// TwinCAT 3 PLC project Untitled1
// ProgramVersion: 3.1.4020.1
// libraries:
//   Tc2_EtherCAT, * (Beckhoff Automation GmbH)
//   Tc2_MC2, * (Beckhoff Automation GmbH)
//   Tc2_NCI, * (Beckhoff Automation GmbH)
//   Tc2_Standard, * (Beckhoff Automation GmbH)
//   Tc2_System, * (Beckhoff Automation GmbH)
//   Tc3_Module, * (Beckhoff Automation GmbH)
// project tree:
//   DUTs/ ST_DOX_Control.TcDUT, ST_DOX_STATUS.TcDUT, ST_FastMFunc.TcDUT, ST_MTO_Input.TcDUT, ST_MTO_Outputs.TcDUT, ST_NciChannelFromPlc.TcDUT, ST_NciChannelToPlc.TcDUT
//   / PlcTask.TcTTO
//   POUs/FB_Initialize Axes/ FB_Initialize.TcPOU, ST_Intern_Initialize.TcDUT, ST_PAIn_Initialize.TcDUT, ST_Status_Initialize.TcDUT, ST_Config_Initialize.TcDUT
//   POUs/FB_Valve/ FB_Valve.TcPOU, ST_Config_Valve.TcDUT, ST_PAIn_Valve.TcDUT, ST_PAOut_Valve.TcDUT
//   POUs/FB_Interpreter/ FB_Interpreter.TcPOU, ST_Config_Interpreter.TcDUT, ST_Intern_Interpreter.TcDUT, ST_PAIn_Interpreter.TcDUT, ST_PAOut_Interpreter.TcDUT, ST_Status_Interpreter.TcDUT
//   POUs/POU_Main/ MAIN.TcPOU, ST_Config_Main.TcDUT, ST_Intern_Main.TcDUT, ST_PAIn_Main.TcDUT, ST_PAOut_Main.TcDUT, ST_Status_Main.TcDUT
//   POUs/POU_Drops/ POU_Drops.TcPOU, ST_Config_Drops.TcDUT, ST_PAIn_Drops.TcDUT, ST_PAOut_Drops.TcDUT
// real-time tasks:
//   TASK PlcTask: cycle T#10ms, priority 20, ADS port 350
// motion (NC):
//   TASK NC-Task 1 SAF: cycle T#2ms, priority 4, ADS port 501
//   TASK NC-Task 1 SVB: cycle T#10ms, priority 8, ADS port 511
//   AXIS Axis 1 (id 1)
//     Dynamic: AccelerationMaximum=700, DecelerationMaximum=700, Acceleration=632.077, Deceleration=632.077, Jerk=142686, DelayTime=0.008, OverrideType=4
//     Velo: RefSync=5, SlowManual=25, FastManual=50, Fast=50, Maximum=280
//     PositionAreaControl: Enable=false, RefSearch=false
//     TargetPosControl: Enable=false
//     OtherSettings: AllowMotionCmdToSlave=true
//     encoder EncType=4
//       EncPara: ScaleFactorNumerator=0.002334, MaxCount=#x0000ffff
//         ActPosCorrection: Time=0.02
//         Inc: RefSearchInverse=true, RefSyncInverse=false, RefMode=1, RefSoftSyncMask=#x0000ffff
//     drive DrvType=24
//       Analog: VeloReferenz=300
//       TimeComp: TaskDelayCycles=1
//     controller CtrType=2
//       CtrPara: PriorControlFactor=1
//         PosDiffControl: Enable=false
//         PID: PosKp=100, PosExtKp=100, DeadBandPosition=0.01
//         Observer: BandWidth=20
//   AXIS Axis 2 (id 2)
//     Dynamic: AccelerationMaximum=700, DecelerationMaximum=700, Acceleration=632.077, Deceleration=632.077, Jerk=142686, DelayTime=0.008, OverrideType=4
//     Velo: RefSync=5, SlowManual=25, FastManual=50, Fast=50, Maximum=280
//     PositionAreaControl: Enable=false, RefSearch=false
//     TargetPosControl: Enable=false
//     OtherSettings: AllowMotionCmdToSlave=true
//     encoder EncType=4
//       EncPara: ScaleFactorNumerator=0.002334, MaxCount=#x0000ffff
//         ActPosCorrection: Time=0.02
//         Inc: RefSearchInverse=true, RefSyncInverse=false, RefMode=1, RefSoftSyncMask=#x0000ffff
//     drive DrvType=24
//       Analog: VeloReferenz=300
//       TimeComp: TaskDelayCycles=1
//     controller CtrType=2
//       CtrPara: PriorControlFactor=1
//         PosDiffControl: Enable=false
//         PID: PosKp=100, PosExtKp=100, DeadBandPosition=0.01
//         Observer: BandWidth=20
// I/O:
//   DEVICE Device 2 (EtherCAT), AmsNetId 192.168.31.63.3.1
//     Term 1 (EK1101) [EK1101 EtherCAT Coupler (2A E-Bus, ID switch)]
//       Term 2 (EL2008) [EL2008 8Ch. Dig. Output 24V, 0.5A]
//       Term 3 (EL7037) [EL7037 1Ch. Stepper motor output stage (24V, 1.5A)]
//       Term 4 (EL7037) [EL7037 1Ch. Stepper motor output stage (24V, 1.5A)]
//       Term 5 (EL1018) [EL1018 8Ch. Dig. Input 24V, 10µs]
//       Term 6 (EL4004) [EL4004 4Ch. Ana. Output 0-10V, 12bit]
//       Term 7 (EL3064) [EL3064 4Ch. Ana. Input 0-10V]
//       Term 8 (EL3318) [EL3318 8Ch. Ana Input Thermocouple (TC)]
//       Term 9 (EL9576) [EL9576 Brake chopper terminal]
//       Term 10 (EL2212) [EL2212 2Ch. dig. output with overexcitation (24V DC, 2.5A, 10A Peak)]
//       Term 11 (EL9011) [EL9011 End Terminal]
// variable links:
//   NC-Task 1 SAF/Axes/Axis 1 <-> Device 2 (EtherCAT)/Term 1 (EK1101)/Term 3 (EL7037)
//     Drive/Inputs/In/nState1 @bit 3 <-> STM Status/Status/Error
//     Drive/Inputs/In/nState1 @bit 7 <-> STM Status/Status/Motor stall
//     Drive/Inputs/In/nState1 @bit 5 <-> STM Status/Status/Moving negative
//     Drive/Inputs/In/nState1 @bit 4 <-> STM Status/Status/Moving positive
//     Drive/Inputs/In/nState1 @bit 1 <-> STM Status/Status/Ready
//     Drive/Inputs/In/nState1 <-> STM Status/Status/Ready to enable
//     Drive/Inputs/In/nState1 @bit 6 <-> STM Status/Status/Torque reduced
//     Drive/Inputs/In/nState1 @bit 2 <-> STM Status/Status/Warning
//     Drive/Inputs/In/nState2 @bit 3 <-> STM Status/Status/Digital input 1
//     Drive/Inputs/In/nState2 @bit 4 <-> STM Status/Status/Digital input 2
//     Drive/Inputs/In/nState2 @bit 5 <-> STM Status/Status/Sync error
//     Drive/Inputs/In/nState2 @bit 7 <-> STM Status/Status/TxPDO Toggle
//     Drive/Inputs/In/nState4 @bit 1 <-> WcState/InputToggle
//     Drive/Inputs/In/nState4 <-> WcState/WcState
//     Drive/Outputs/Out/nCtrl1 <-> STM Control/Control/Enable
//     Drive/Outputs/Out/nCtrl1 @bit 2 <-> STM Control/Control/Reduce torque
//     Drive/Outputs/Out/nCtrl1 @bit 1 <-> STM Control/Control/Reset
//     Drive/Outputs/Out/nCtrl2 @bit 3 <-> STM Control/Control/Digital output 1
//     Drive/Outputs/Out/nDataOut2[0] <-> STM Velocity/Velocity
//     Enc/Inputs/In/nDataIn1[0] <-> ENC Status compact/Counter value
//     Enc/Inputs/In/nDataIn2[0] <-> ENC Status compact/Latch value
//     Enc/Inputs/In/nState1 @bit 4 <-> ENC Status compact/Status/Counter overflow
//     Enc/Inputs/In/nState1 @bit 3 <-> ENC Status compact/Status/Counter underflow
//     Enc/Inputs/In/nState1 @bit 7 <-> ENC Status compact/Status/Extrapolation stall
//     Enc/Inputs/In/nState1 <-> ENC Status compact/Status/Latch C valid
//     Enc/Inputs/In/nState1 @bit 1 <-> ENC Status compact/Status/Latch extern valid
//     Enc/Inputs/In/nState1 @bit 2 <-> ENC Status compact/Status/Set counter done
//     Enc/Inputs/In/nState2 @bit 4 <-> ENC Status compact/Status/Status of extern latch
//     Enc/Inputs/In/nState2 <-> ENC Status compact/Status/Status of input A
//     Enc/Inputs/In/nState2 @bit 1 <-> ENC Status compact/Status/Status of input B
//     Enc/Inputs/In/nState2 @bit 2 <-> ENC Status compact/Status/Status of input C
//     Enc/Inputs/In/nState2 @bit 5 <-> ENC Status compact/Status/Sync error
//     Enc/Inputs/In/nState2 @bit 7 <-> ENC Status compact/Status/TxPDO Toggle
//     Enc/Inputs/In/nState4 @bit 1 <-> WcState/InputToggle
//     Enc/Inputs/In/nState4 <-> WcState/WcState
//     Enc/Outputs/Out/nCtrl1 <-> ENC Control compact/Control/Enable latch C
//     Enc/Outputs/Out/nCtrl1 @bit 3 <-> ENC Control compact/Control/Enable latch extern on negative edge
//     Enc/Outputs/Out/nCtrl1 @bit 1 <-> ENC Control compact/Control/Enable latch extern on positive edge
//     Enc/Outputs/Out/nCtrl1 @bit 2 <-> ENC Control compact/Control/Set counter
//     Enc/Outputs/Out/nDataOut1[0] <-> ENC Control compact/Set counter value
//   NC-Task 1 SAF/Axes/Axis 2 <-> Device 2 (EtherCAT)/Term 1 (EK1101)/Term 4 (EL7037)
//     Drive/Inputs/In/nState1 @bit 3 <-> STM Status/Status/Error
//     Drive/Inputs/In/nState1 @bit 7 <-> STM Status/Status/Motor stall
//     Drive/Inputs/In/nState1 @bit 5 <-> STM Status/Status/Moving negative
//     Drive/Inputs/In/nState1 @bit 4 <-> STM Status/Status/Moving positive
//     Drive/Inputs/In/nState1 @bit 1 <-> STM Status/Status/Ready
//     Drive/Inputs/In/nState1 <-> STM Status/Status/Ready to enable
//     Drive/Inputs/In/nState1 @bit 6 <-> STM Status/Status/Torque reduced
//     Drive/Inputs/In/nState1 @bit 2 <-> STM Status/Status/Warning
//     Drive/Inputs/In/nState2 @bit 3 <-> STM Status/Status/Digital input 1
//     Drive/Inputs/In/nState2 @bit 4 <-> STM Status/Status/Digital input 2
//     Drive/Inputs/In/nState2 @bit 5 <-> STM Status/Status/Sync error
//     Drive/Inputs/In/nState2 @bit 7 <-> STM Status/Status/TxPDO Toggle
//     Drive/Inputs/In/nState4 @bit 1 <-> WcState/InputToggle
//     Drive/Inputs/In/nState4 <-> WcState/WcState
//     Drive/Outputs/Out/nCtrl1 <-> STM Control/Control/Enable
//     Drive/Outputs/Out/nCtrl1 @bit 2 <-> STM Control/Control/Reduce torque
//     Drive/Outputs/Out/nCtrl1 @bit 1 <-> STM Control/Control/Reset
//     Drive/Outputs/Out/nCtrl2 @bit 3 <-> STM Control/Control/Digital output 1
//     Drive/Outputs/Out/nDataOut2[0] <-> STM Velocity/Velocity
//     Enc/Inputs/In/nDataIn1[0] <-> ENC Status compact/Counter value
//     Enc/Inputs/In/nDataIn2[0] <-> ENC Status compact/Latch value
//     Enc/Inputs/In/nState1 @bit 4 <-> ENC Status compact/Status/Counter overflow
//     Enc/Inputs/In/nState1 @bit 3 <-> ENC Status compact/Status/Counter underflow
//     Enc/Inputs/In/nState1 @bit 7 <-> ENC Status compact/Status/Extrapolation stall
//     Enc/Inputs/In/nState1 <-> ENC Status compact/Status/Latch C valid
//     Enc/Inputs/In/nState1 @bit 1 <-> ENC Status compact/Status/Latch extern valid
//     Enc/Inputs/In/nState1 @bit 2 <-> ENC Status compact/Status/Set counter done
//     Enc/Inputs/In/nState2 @bit 4 <-> ENC Status compact/Status/Status of extern latch
//     Enc/Inputs/In/nState2 <-> ENC Status compact/Status/Status of input A
//     Enc/Inputs/In/nState2 @bit 1 <-> ENC Status compact/Status/Status of input B
//     Enc/Inputs/In/nState2 @bit 2 <-> ENC Status compact/Status/Status of input C
//     Enc/Inputs/In/nState2 @bit 5 <-> ENC Status compact/Status/Sync error
//     Enc/Inputs/In/nState2 @bit 7 <-> ENC Status compact/Status/TxPDO Toggle
//     Enc/Inputs/In/nState4 @bit 1 <-> WcState/InputToggle
//     Enc/Inputs/In/nState4 <-> WcState/WcState
//     Enc/Outputs/Out/nCtrl1 <-> ENC Control compact/Control/Enable latch C
//     Enc/Outputs/Out/nCtrl1 @bit 3 <-> ENC Control compact/Control/Enable latch extern on negative edge
//     Enc/Outputs/Out/nCtrl1 @bit 1 <-> ENC Control compact/Control/Enable latch extern on positive edge
//     Enc/Outputs/Out/nCtrl1 @bit 2 <-> ENC Control compact/Control/Set counter
//     Enc/Outputs/Out/nDataOut1[0] <-> ENC Control compact/Set counter value
//   Untitled1/Untitled1 Instance <-> Device 2 (EtherCAT)/Term 1 (EK1101)/Term 10 (EL2212)
//     PlcTask Inputs/MAIN.stPAIn/stPAInDrops/stValve/stDOXStatus1/bError <-> DOX Status (MTO) Channel 1/Status/Error
//     PlcTask Inputs/MAIN.stPAIn/stPAInDrops/stValve/stDOXStatus1/bPWMActive <-> DOX Status (MTO) Channel 1/Status/PWM active
//     PlcTask Inputs/MAIN.stPAIn/stPAInDrops/stValve/stDOXStatus1/bReadyToActivate <-> DOX Status (MTO) Channel 1/Status/Ready to activate
//     PlcTask Inputs/MAIN.stPAIn/stPAInDrops/stValve/stDOXStatus1/bTxPDO <-> DOX Status (MTO) Channel 1/Status/TxPDO Toggle
//     PlcTask Inputs/MAIN.stPAIn/stPAInDrops/stValve/stDOXStatus1/bWarning <-> DOX Status (MTO) Channel 1/Status/Warning
//     PlcTask Inputs/MAIN.stPAIn/stPAInDrops/stValve/stMTOInputs1/b2InputCycleCounter <-> MTO Inputs Channel 1/Status/Input cycle counter
//     PlcTask Inputs/MAIN.stPAIn/stPAInDrops/stValve/stMTOInputs1/bOutputBufferOverflow <-> MTO Inputs Channel 1/Status/Output buffer overflow
//     PlcTask Inputs/MAIN.stPAIn/stPAInDrops/stValve/stMTOInputs1/bOutputShortCircuit <-> MTO Inputs Channel 1/Status/Output short circuit
//     PlcTask Inputs/MAIN.stPAIn/stPAInDrops/stValve/stMTOInputs1/bOutputState <-> MTO Inputs Channel 1/Status/Output state
//     PlcTask Inputs/MAIN.stPAIn/stPAInDrops/stValve/stMTOInputs1/bWarning <-> MTO Inputs Channel 1/Status/Warning
//     PlcTask Inputs/MAIN.stPAIn/stPAInDrops/stValve/stMTOInputs1/iEventsInOutput <-> MTO Inputs Channel 1/Status/Events in output buffer
//     PlcTask Inputs/MAIN.stPAIn/stPAInDrops/stValve/stMTOInputs1/iOutputOrderFeedback <-> MTO Inputs Channel 1/Status/Output order feedback
//     PlcTask Outputs/MAIN.stPAOut/stPAOutDrops/stValve/stDoxControl1/bPWM <-> DOX Control (MTO) Channel 1/Control/PWM
//     PlcTask Outputs/MAIN.stPAOut/stPAOutDrops/stValve/stDoxControl1/bReset <-> DOX Control (MTO) Channel 1/Control/Reset
//     PlcTask Outputs/MAIN.stPAOut/stPAOutDrops/stValve/stMTOOutputs1/bBufferReset <-> MTO Outputs 2x Channel 1/Ctrl/Output buffer reset
//     PlcTask Outputs/MAIN.stPAOut/stPAOutDrops/stValve/stMTOOutputs1/bEnableManualOp <-> MTO Outputs 2x Channel 1/Ctrl/Enable manual operation
//     PlcTask Outputs/MAIN.stPAOut/stPAOutDrops/stValve/stMTOOutputs1/bForceOrder <-> MTO Outputs 2x Channel 1/Ctrl/Force order
//     PlcTask Outputs/MAIN.stPAOut/stPAOutDrops/stValve/stMTOOutputs1/bManualOutputState <-> MTO Outputs 2x Channel 1/Ctrl/Manual output state
//     PlcTask Outputs/MAIN.stPAOut/stPAOutDrops/stValve/stMTOOutputs1/bOutputEventState1 <-> MTO Outputs 2x Channel 1/Outputs/Output event state 1
//     PlcTask Outputs/MAIN.stPAOut/stPAOutDrops/stValve/stMTOOutputs1/bOutputEventState2 <-> MTO Outputs 2x Channel 1/Outputs/Output event state 2
//     PlcTask Outputs/MAIN.stPAOut/stPAOutDrops/stValve/stMTOOutputs1/iNoOfOutputEvents <-> MTO Outputs 2x Channel 1/Ctrl/No of output events
//     PlcTask Outputs/MAIN.stPAOut/stPAOutDrops/stValve/stMTOOutputs1/iOutputOrderCount <-> MTO Outputs 2x Channel 1/Ctrl/Output order counter
//     PlcTask Outputs/MAIN.stPAOut/stPAOutDrops/stValve/stMTOOutputs1/tOutputEventTime1 <-> MTO Outputs 2x Channel 1/Output event time 1
//     PlcTask Outputs/MAIN.stPAOut/stPAOutDrops/stValve/stMTOOutputs1/tOutputEventTime2 <-> MTO Outputs 2x Channel 1/Output event time 2
//   Untitled1/Untitled1 Instance <-> Device 2 (EtherCAT)/Term 1 (EK1101)/Term 3 (EL7037)
//     PlcTask Inputs/MAIN.stPAIn/stInit/bXCam <-> STM Status/Status/Digital input 1
//   Untitled1/Untitled1 Instance <-> Device 2 (EtherCAT)/Term 1 (EK1101)/Term 4 (EL7037)
//     PlcTask Inputs/MAIN.stPAIn/stInit/bYCam <-> STM Status/Status/Digital input 1
//   Untitled1/Untitled1 Instance <-> NC-Task 1 SAF/Axes/Axis 1
//     PlcTask Inputs/MAIN.fbInitialize.XAxis.NcToPlc <-> Outputs/ToPlc
//     PlcTask Outputs/MAIN.fbInitialize.XAxis.PlcToNc <-> Inputs/FromPlc
//   Untitled1/Untitled1 Instance <-> NC-Task 1 SAF/Axes/Axis 2
//     PlcTask Inputs/MAIN.fbInitialize.YAxis.NcToPlc <-> Outputs/ToPlc
//     PlcTask Outputs/MAIN.fbInitialize.YAxis.PlcToNc <-> Inputs/FromPlc
//   Untitled1/Untitled1 Instance <-> NC-Task 1 SAF/Channel 2
//     PlcTask Inputs/MAIN.stPAIn/stInterp/in_stItpToPlc <-> Outputs/ToPlc
//     PlcTask Inputs/MAIN.stPAIn/stMBits <-> Outputs/ToPlc/FastMFuncMask[1]
//     PlcTask Outputs/MAIN.stPAOut/stInterp/out_stPlcToItp <-> Inputs/FromPlc

CONFIGURATION Untitled1
    RESOURCE PLC ON TwinCAT3
        TASK PlcTask(INTERVAL := T#10ms, PRIORITY := 20);
        PROGRAM MAIN WITH PlcTask : MAIN;
    END_RESOURCE
END_CONFIGURATION

// ---- DUTs/ST_DOX_Control.TcDUT
TYPE ST_DOX_Control :
STRUCT
	bBit0    :				BIT;	//71.0
	bBit1    :				BIT;
	bBit2    :				BIT;
	bPWM  :					BIT:=1;	//71.3
	bBit4  :				BIT;
	bBit5  :				BIT;
	bBit6  :				BIT;
	bReset  :				BIT;	//71.7
	BByte8   :				BYTE;
	
END_STRUCT
END_TYPE

// ---- DUTs/ST_DOX_STATUS.TcDUT
TYPE ST_DOX_STATUS :
STRUCT
	bReadyToActivate:	BIT;
	bPWMActive:			BIT;
	bWarning:			BIT;
	bError:				BIT;
	bTxPDO:				BIT;
END_STRUCT
END_TYPE

// ---- DUTs/ST_FastMFunc.TcDUT
TYPE ST_FastMFunc :
STRUCT
	bMbit0:			BIT;
	bMBit1:			BIT;
	bMBit2:			BIT;
	bMBit3:			BIT;
	bMBit4:			BIT;
	bMBit5:			BIT;
	bMBit6:			BIT;
	bMBit7:			BIT;
	bMBit8:			BIT;
	bMBit9:			BIT;
	bMBit10:		BIT;
	bMBit11:		BIT;
	bMBit12:		BIT;
	bMBit13:		BIT;
	bMBit14:		BIT;
	bMBit15:		BIT;
	bMBit16:		BIT;
	bMBit17:		BIT;
	bMBit18:		BIT;
	bMBit19:		BIT;
	bMBit20:		BIT;
	bMBit21:		BIT;
	bMBit22:		BIT;
	bMBit23:		BIT;
	bMBit24:		BIT;
	bMBit25:		BIT;
	bMBit26:		BIT;
	bMBit27:		BIT;
	bMBit28:		BIT;
	bMBit29:		BIT;
	bMBit30:		BIT;
	bMBit31:		BIT;	
END_STRUCT
END_TYPE

// ---- DUTs/ST_MTO_Input.TcDUT
TYPE ST_MTO_Input :
STRUCT
	bOutputShortCircuit:			BOOL;
	bOutputBufferOverflow:			BOOL;
	bOutputState:					BOOL;
	bWarning:						BOOL;
	b2InputCycleCounter:			BOOL;
	iOutputOrderFeedback:			USINT;
	iEventsInOutput:				USINT;
END_STRUCT
END_TYPE

// ---- DUTs/ST_MTO_Outputs.TcDUT
TYPE ST_MTO_Outputs :
STRUCT
	
	bBufferReset    :				BIT;	//73.0
	bManualOutputState    :			BIT;
	bForceOrder    :				BIT:=1;
	bEnableManualOp  :				BIT;	//73.3
	bBit4  :						BIT;
	bBit5  :						BIT;
	bBit6  :						BIT;
	bBit7  :						BIT;
	iOutputOrderCount  :			USINT;	//74.0
	iNoOfOutputEvents  :			USINT;	//75.0
	Bbyte24:						BYTE;
	bOutputEventState1	:			BIT;
	bOutputEventState2	:			BIT;
	tOutputEventTime1:				UDINT;
	tOutputEventTime2:				UDINT;
END_STRUCT
END_TYPE

// ---- DUTs/ST_NciChannelFromPlc.TcDUT
TYPE ST_NciChannelFromPlc :
STRUCT
    nSkipLine        : WORD; (* Mask to skip lines *)
    nItpMode         : WORD;
    nMFuncGranted    : WORD; (* granted signal of the M-function *)
    nReserved1       : ARRAY[7..8] OF BYTE;
    nChaAxesOvr      : DWORD; (* Channel override in percent * 100 *)
    nChaSpindleOvr   : DWORD;
    nReserved2       : ARRAY[17..128] OF BYTE;
END_STRUCT
END_TYPE

// ---- DUTs/ST_NciChannelToPlc.TcDUT
TYPE ST_NciChannelToPlc :
STRUCT
	
    nJobNo         : DWORD;
    nFastMFuncMask : ARRAY[1..5] OF DWORD; (* Mask to evaluate fast M-functions *)
    nHskMFuncNo    : WORD; (* evaluate M-function with handshake *)
    nHskMFuncReq   : WORD;
    nHFuncValue    : DINT;
    nSpindleRpm    : WORD;
    nTool          : WORD;
    nReserved1     : ARRAY[37..132] OF BYTE;
    nLoadedProg    : DWORD; (* loaded program number if exist *)
    nItpMode       : WORD; (* Interpreter mode *)
    nItpState      : WORD; (* Interpreter status *)
    nItpErrCode    : UDINT; (* Interpreter-Channel Error Code Changed from *WORD*)
    nReserved2     : ARRAY[143..150] OF BYTE;
	
END_STRUCT
END_TYPE

// ---- POUs/FB_Initialize Axes/ST_Intern_Initialize.TcDUT
TYPE ST_Intern_Initialize :
STRUCT
		tnReady		:TON;
		
END_STRUCT
END_TYPE

// ---- POUs/FB_Initialize Axes/ST_PAIn_Initialize.TcDUT
TYPE ST_PAIn_Initialize :
STRUCT
	
(*Homing Notches*)	
	bXCam	:BOOL;  	
	bYCam	:BOOL;
	
END_STRUCT
END_TYPE

// ---- POUs/FB_Initialize Axes/ST_Status_Initialize.TcDUT
TYPE ST_Status_Initialize :
STRUCT
	bFini	:BOOL;
	bBus	:BOOL;
	bErr	:BOOL;
	nErr	:UDINT;
	iItpState:	UDINT;
	iState: INT;
END_STRUCT
END_TYPE

// ---- POUs/FB_Initialize Axes/ST_Config_Initialize.TcDUT
TYPE ST_Config_Initialize :
STRUCT
	nXA					:UDINT:=1;
	nYA					:UDINT:=2;
	nZA					:UDINT:=0;
	nGroup				:UDINT:=3;
	tTimeO				:TIME:=T#5S;
	g_strProgram		:STRING := 'C:\Users\Furkan\Desktop\FirstNciSample\TestIt.nc';
	bExe				:BOOL:=TRUE;
	bSta				:BOOL:=TRUE;
	bSto				:BOOL:=FALSE;
	
END_STRUCT
END_TYPE

// ---- POUs/FB_Valve/ST_Config_Valve.TcDUT
TYPE ST_Config_Valve:
STRUCT
END_STRUCT
END_TYPE

// ---- POUs/FB_Valve/ST_PAIn_Valve.TcDUT
TYPE ST_PAIn_Valve :
STRUCT
	stDOXStatus1: ST_DOX_STATUS;
	
	stMTOInputs1: ST_MTO_Input;
	
	
	

END_STRUCT
END_TYPE

// ---- POUs/FB_Valve/ST_PAOut_Valve.TcDUT
TYPE ST_PAOut_Valve :
STRUCT
	stMTOOutputs1:			ST_MTO_Outputs;
	stDoxControl1:			ST_DOX_Control;
	
	
	
END_STRUCT
END_TYPE

// ---- POUs/FB_Interpreter/ST_Config_Interpreter.TcDUT
TYPE ST_Config_Interpreter :
STRUCT
	bInit				:BOOL;
	nXA					:UDINT:=1;
	nYA					:UDINT:=2;
	nZA					:UDINT:=0;
	nGroup				:UDINT:=3;
	tTimeO				:TIME:=T#5S;
	g_strProgram		:STRING := 'D:\Semester\NC.nc';
	bExe				:BOOL:=TRUE;
	bSta				:BOOL:=TRUE;
	bSto				:BOOL:=FALSE;
	
END_STRUCT
END_TYPE

// ---- POUs/FB_Interpreter/ST_Intern_Interpreter.TcDUT
TYPE ST_Intern_Interpreter :
STRUCT
	
		
END_STRUCT
END_TYPE

// ---- POUs/FB_Interpreter/ST_PAIn_Interpreter.TcDUT
TYPE ST_PAIn_Interpreter :
STRUCT

		in_stItpToPlc			:NCTOPLC_NCICHANNEL_REF;
	
END_STRUCT
END_TYPE

// ---- POUs/FB_Interpreter/ST_PAOut_Interpreter.TcDUT
TYPE ST_PAOut_Interpreter :
STRUCT
	
	
	out_stPlcToItp			:PLCTONC_NCICHANNEL_REF;	
END_STRUCT
END_TYPE

// ---- POUs/FB_Interpreter/ST_Status_Interpreter.TcDUT
TYPE ST_Status_Interpreter :
STRUCT
	bFini	:BOOL;
	bBus	:BOOL;
	bErr	:BOOL;
	nErr	:UDINT;
	iItpState:	UDINT;
	iState: INT;
END_STRUCT
END_TYPE

// ---- POUs/POU_Main/ST_Config_Main.TcDUT
TYPE ST_Config_Main :
STRUCT
	
	stInterp			:ST_Config_Interpreter;
	stInit				:ST_Config_Initialize;
END_STRUCT
END_TYPE

// ---- POUs/POU_Main/ST_Intern_Main.TcDUT
TYPE ST_Intern_Main :
STRUCT
	count: INT;
	
END_STRUCT
END_TYPE

// ---- POUs/POU_Main/ST_PAIn_Main.TcDUT
TYPE ST_PAIn_Main :
STRUCT
	(* stNcToPlc	:ST_NciChannelToPlc;  
	stNciIn		:ST_NCInterpreter_PAIn;*)

	stInit			:ST_PAIn_Initialize;
	stInterp		:ST_PAIn_Interpreter;
	stMBits			:ST_FastMFunc;
	stPAInDrops		:ST_PAIn_Drops;
	

END_STRUCT
END_TYPE

// ---- POUs/POU_Main/ST_PAOut_Main.TcDUT
TYPE ST_PAOut_Main :
STRUCT
	
	stInterp					:ST_PAOut_Interpreter;
	stPAOutDrops				:ST_PAOut_Drops;
END_STRUCT
END_TYPE

// ---- POUs/POU_Main/ST_Status_Main.TcDUT
TYPE ST_Status_Main :
STRUCT
	stInterp				:ST_Status_Interpreter;
	stInit					:ST_Status_Initialize;
END_STRUCT
END_TYPE

// ---- POUs/POU_Drops/ST_Config_Drops.TcDUT
TYPE ST_Config_Drops :
STRUCT
	stValve: ST_Config_Valve;
	
END_STRUCT
END_TYPE

// ---- POUs/POU_Drops/ST_PAIn_Drops.TcDUT
TYPE ST_PAIn_Drops :
STRUCT
	stValve 			:ST_PAIn_Valve;
	
END_STRUCT
END_TYPE

// ---- POUs/POU_Drops/ST_PAOut_Drops.TcDUT
TYPE ST_PAOut_Drops :
STRUCT
	stValve: ST_PAOut_Valve;
	
END_STRUCT
END_TYPE

// ---- POUs/POU_Main/MAIN.TcPOU
PROGRAM MAIN

VAR
	stIntern			:ST_Intern_Main;
	fbInitialize		:FB_Initialize;
	fbInterpreter		:FB_Interpreter;
	stStatus			:ST_Status_Main;
	iState				:INT;
END_VAR

VAR_INPUT
	stConfig			:ST_Config_Main;
	stPAIn	AT%I*		:ST_PAIn_Main;
	
END_VAR

VAR_OUTPUT
	stPAOut	AT%Q*		:ST_PAOut_Main;
	
END_VAR

fbInitialize(stPAIn:=stPAIn.stInit,
			stConfig:=stConfig.stInit,
			stStatus=>stStatus.stInit	);


fbInterpreter(stConfig:=stConfig.stInterp,
				stPAOut=>stPAOut.stInterp,
				stStatus=>stStatus.stInterp);

fbInterpreter.stPAIn.in_stItpToPlc:=stPAIn.stInterp.in_stItpToPlc;	


CASE iState OF
	
		00: fbInitialize.bExec:=TRUE;
	
		IF NOT fbInitialize.bBus THEN
			IF fbInitialize.bFini THEN 
				iState:=10;
			END_IF
		END_IF
		
		10: fbInterpreter.bExec:=TRUE;
	
		IF NOT fbInterpreter.bBus THEN
			IF fbInterpreter.bFini THEN 
				iState:=20;
			END_IF
		END_IF
		
	
END_CASE

END_PROGRAM

// ---- POUs/FB_Initialize Axes/FB_Initialize.TcPOU
FUNCTION_BLOCK FB_Initialize
VAR_INPUT
	stPAIn	 				:ST_PAIn_Initialize;
	stConfig				:ST_Config_Initialize;
	bExec				:BOOL;
END_VAR
	
VAR_OUTPUT
	bFini	:BOOL;
	bBus	:BOOL;
	bErr	:BOOL;

	stStatus				:ST_Status_Initialize;
END_VAR

VAR
	stIntern				:ST_Intern_Initialize;
	(*Axis References*)
	XAxis					:AXIS_REF;
	YAxis					:AXIS_REF;
	(*Motion Control Definitions*)
	fbPower_X				:MC_Power;
	fbPower_Y				:MC_Power;
	fbHome_X				:MC_Home;
	fbHome_Y				:MC_Home;
	fbBuildGrp				:CfgBuildExt3DGroup;
END_VAR


XAxis.ReadStatus();
YAxis.ReadStatus();
fbPower_X(Axis:=XAxis);
fbPower_Y(Axis:=YAxis);	
fbHome_X(Axis:=XAxis);
fbHome_Y(Axis:=YAxis);	

CASE stStatus.iState OF 

	00:	IF bExec THEN
			bBus:=TRUE;
 			stStatus.iState:=05;
		END_IF
		

05:
(*Enable X-Axis*)
		fbPower_X.Enable			:=TRUE;
		fbPower_X.Enable_Positive	:=TRUE;
		fbPower_X.Enable_Negative	:=TRUE;
		
(*Enable Y-Axis*)

		fbPower_Y.Enable			:=TRUE;
		fbPower_Y.Enable_Positive	:=TRUE;
		fbPower_Y.Enable_Negative	:=TRUE;
		
	stIntern.tnReady(IN:=fbPower_X.Status AND fbPower_Y.Status,PT:=T#100MS);
			
		IF stIntern.tnReady.Q THEN
			stStatus.iState:=10;
		END_IF
10:	(*Home X-Axis*)
		fbHome_X.HomingMode			:=MC_DefaultHoming;
		fbHome_X.bCalibrationCam	:=stPAIn.bXCam;
		fbHome_X.Execute			:= stConfig.bExe;
		fbHome_X.Position			:= 0;
	(*Home Y-Axis*)
		fbHome_Y.HomingMode			:=MC_DefaultHoming;
		fbHome_Y.bCalibrationCam	:=stPAIn.bYCam;
		fbHome_Y.Execute			:= stConfig.bExe;
		fbHome_Y.Position			:= 0;
		
		IF NOT fbHome_X.Error AND NOT fbHome_Y.Error AND fbHome_X.Done AND fbHome_Y.Done THEN
			stStatus.iState:=20;
		END_IF
		
20:	(* Build group for interpolation*)
		fbBuildGrp	(
		bExecute	:= TRUE ,
		nGroupId	:= stConfig.nGroup,
		nXAxisId	:= stConfig.nXA,
		nYAxisId	:= stConfig.nYA,
		nZAxisId	:= stConfig.nZA,
		nQ1AxisId	:= 0,
		nQ2AxisId	:= 0,
		nQ3AxisId	:= 0,
		nQ4AxisId	:= 0,
		nQ5AxisId	:= 0,
		tTimeOut	:= T#200MS,
		bErr		=>stStatus.bErr,
		bBusy		=>stStatus.bBus,
		nErrId		=>stStatus.nErr);	
				
	stIntern.tnReady(IN:=TRUE AND NOT stStatus.bErr ,PT:=T#2S);
	IF stIntern.tnReady.Q THEN
		bFini:=TRUE;
		bBus:=FALSE;
		stStatus.iState:=30;
	END_IF		

END_CASE

END_FUNCTION_BLOCK

// ---- POUs/FB_Interpreter/FB_Interpreter.TcPOU
FUNCTION_BLOCK FB_Interpreter
VAR
	fbLoadProg				:ItpLoadProgEx;
	fbStart					:ItpStartStopEx;
END_VAR
VAR_INPUT
	bExec					:BOOL;
	stPAIn					:ST_PAIn_Interpreter;
	stConfig				:ST_Config_Interpreter;
END_VAR
VAR_OUTPUT
	bFini	:BOOL;
	bBus	:BOOL;
	bErr	:BOOL;

	stPAOut					:ST_PAOut_Interpreter;
	stStatus				:ST_Status_Interpreter;
END_VAR

CASE stStatus.iState OF
		

	00: IF 	bExec THEN
			bBus:=TRUE;
			stStatus.iState:=05;
		END_IF


	05:
		fbLoadProg(
		bExecute	:= TRUE,
		sPrg		:= stConfig.g_strProgram,
		nLength		:= LEN(stConfig.g_strProgram),
		tTimeOut	:= T#200MS,
		sNciToPlc	:= MAIN.stPAIn.stInterp.in_stItpToPlc);
		
	stStatus.iItpState		:=	ItpGetStateInterpreter(stPAIn.in_stItpToPlc );
	
	IF stStatus.iItpState = NCI_INTERPRETER_READY THEN
		(* load part program succeeded *)
		stStatus.iState	:= 10;
	ELSIF stStatus.iItpState = NCI_INTERPRETER_ABORTED THEN
		(* load program failed - probably there is a load time error, e.g. syntax error *)
		(* add error handling here *)
		stStatus.bErr		:= TRUE;
		stStatus.nErr	:= 4711;	(* substitute with own error code *)
		stStatus.iState	:= 200;
	END_IF
	
	10: ItpSetOverridePercent( fOverridePercent:=100, sPlcToNci:=stPAOut.out_stPlcToItp );
	
		fbStart(
				bStart		:= stConfig.bSta,
				bStop		:= stConfig.bSto,
				tTimeOut	:= T#200MS,
				sNciToPlc	:=Main.stPAIn.stInterp.in_stItpToPlc
				);

	IF NOT fbStart.bBusy THEN
		fbStart( bStart:=FALSE, sNciToPlc:=stPAIn.in_stItpToPlc );
		IF NOT fbStart.bErr THEN
			stStatus.iState	:= 20;
		ELSE
			(* an error occured *)
			stStatus.bErr		:= TRUE;
			stStatus.nErr	:= fbStart.nErrId;
			stStatus.iState	:= 200;
		END_IF
	END_IF
		
	20:	stStatus.iItpState	:=	ItpGetStateInterpreter(  sNciToPlc:=MAIN.stPAIn.stInterp.in_stItpToPlc );
	IF stStatus.iItpState <> NCI_INTERPRETER_READY THEN
		bFini:=TRUE;
		bBus:=FALSE;
		stStatus.iState	:= 40;
	END_IF
				
END_CASE

END_FUNCTION_BLOCK

// ---- POUs/FB_Valve/FB_Valve.TcPOU
FUNCTION_BLOCK FB_Valve
VAR_INPUT
	
	stConfig:	ST_Config_Valve;
	stPAIn	:	ST_PAIn_Valve;
	
	iPeriod: 	UDINT:= 40000000;
	tPeriod: 	TIME;
	iDuration: 	UDINT:= 9000000;
	bActivate: 	BOOL:=TRUE;
	
END_VAR
VAR_OUTPUT
	stPAOut	:	ST_PAOut_Valve;
END_VAR
	
VAR
	iEvent1: 		UDINT;
	iEvent2:		UDINT;	
	nNoOfOutputEvents: INT;
	nOutputOrderCnt: USINT;
	
	tnHalt: 			TON;
 	iCurrentTime:  	ULINT;
 	iCurrentTime32:  	UDINT;
	
	nScheduleNo: INT;
	iState:			UINT:=0;
	iLastTime: UDINT;
END_VAR

	iCurrentTime := F_GetCurDcTaskTime64();
	iCurrentTime32:=ULINT_TO_UDINT(iCurrentTime AND 16#FFFFFFFF); 
	
CASE iState OF

0:	
	stPAOut.stMTOOutputs1.bBufferReset:=TRUE;
	iState:=iState+1;

1:
	stPAOut.stMTOOutputs1.bBufferReset:=FALSE;
	iState:=iState+1;
		
2:
	IF stPAIn.stDOXStatus1.bReadyToActivate THEN 
	iState:=10;
	iLastTime:=iCurrentTime32+100000000;
	END_IF

10:
	
	
	iEvent1:=(iLastTime+iPeriod) ; 
	iEvent2:=(iEvent1+iDuration)  ; 
	iLastTime:=iEvent1;	 

	stPAOut.stMTOOutputs1.tOutputEventTime1:=iEvent1;
	stPAOut.stMTOOutputs1.tOutputEventTime2:=iEvent2;	
	stPAOut.stMTOOutputs1.bOutputEventState1:=1;
	stPAOut.stMTOOutputs1.bOutputEventState2:=0;

	iState:=20;
(*10:
	iEvent1:=(iCurrentTime32+iPeriod) MOD 2147483648 ; 
	iEvent2:=(iEvent1+iDuration) MOD 2147483648 ; 
	
	
	iLastTime:=iEvent1;	 
	
	iState:=20; *)
20: 
IF nScheduleNo=3 THEN 
	nScheduleNo := 0;
	nOutputOrderCnt:=stPAIn.stMTOInputs1.iOutputOrderFeedback+1;
	iState:=30;
ELSE
	nScheduleNo := nScheduleNo + 1; 
END_IF 

30:
	IF nScheduleNo=3 THEN 
	nScheduleNo := 0;
	IF NOT INT_TO_BOOL(MAIN.stPAIn.stPAInDrops.stValve.stMTOInputs1.iEventsInOutput) THEN
		iState:=10;
	END_IF
	ELSE
	nScheduleNo := nScheduleNo + 1; 
	END_IF 


END_CASE

stPAOut.stMTOOutputs1.tOutputEventTime1:=iEvent1;
stPAOut.stMTOOutputs1.tOutputEventTime2:=iEvent2;	


stPAOut.stMTOOutputs1.bOutputEventState1:=1;
stPAOut.stMTOOutputs1.bOutputEventState2:=0;

stPAOut.stMTOOutputs1.iNoOfOutputEvents:=2;
stPAOut.stMTOOutputs1.iOutputOrderCount:=nOutputOrderCnt;

END_FUNCTION_BLOCK

// ---- POUs/POU_Drops/POU_Drops.TcPOU
PROGRAM POU_Drops
VAR
	fbValve				:FB_Valve;
	
END_VAR
VAR_INPUT
	stConfig			:ST_Config_Drops;
	stPAInDrops			:ST_PAIn_Drops;
	
END_VAR
VAR_OUTPUT
	stPAOutDrops				:ST_PAOut_Drops;
END_VAR
VAR
	
	
END_VAR

IF MAIN.stPAIn.stMBits.bMBit10 THEN
	
fbValve(stPAIn:=stPAInDrops.stValve,
		stConfig:=stConfig.stValve,
		stPaOut=>stPAOutDrops.stValve);

END_IF

END_PROGRAM
